{attribute 'GeneratedUsingTerminal: EL3314-0030-0021'}
{attribute addProperty BoxType "EL3314-0030-0021"}
{attribute addProperty Id "TC_Inputs_Channel_1AT %I*TC_Inputs_Channel_204FE7509TC_Inputs_Channel_2AT %I*TC_Inputs_Channel_204FE7509TC_Inputs_Channel_3AT %I*TC_Inputs_Channel_204FE7509TC_Inputs_Channel_4AT %I*TC_Inputs_Channel_204FE7509WcStateAT %I*WcState_9091E0EB2InfoDataAT %I*InfoData_94A18F5E2"}
{attribute addProperty CRC "237167355"}
{attribute addProperty Size "40"}
TYPE EL3314_0E22E2FB EXTENDS EtcSlaveTerminalBase_947E5A46 :
STRUCT
	{attribute addProperty Name "TC_Inputs_Channel_1"}
	TC_Inputs_Channel_1 : TC_Inputs_Channel_204FE750;
	{attribute addProperty Name "TC_Inputs_Channel_2"}
	TC_Inputs_Channel_2 : TC_Inputs_Channel_204FE750;
	{attribute addProperty Name "TC_Inputs_Channel_3"}
	TC_Inputs_Channel_3 : TC_Inputs_Channel_204FE750;
	{attribute addProperty Name "TC_Inputs_Channel_4"}
	TC_Inputs_Channel_4 : TC_Inputs_Channel_204FE750;
	{attribute addProperty Name "WcState"}
	WcState : WcState_9091E0EB;
	{attribute addProperty Name "InfoData"}
	InfoData : InfoData_94A18F5E;
END_STRUCT
END_TYPE

(* stored: Version 1.2.0.0, ProductVersion 3.1.4024.9
   DUT EL3314_0E22E2FB: Id {6bb66c0c-989e-4fe7-af5f-82a3cdcbb2d3} *)
